TYPE ST_St020_HMI_IN_OUT : // EXTENDS ST_HMI_TR_CMD :
STRUCT
END_STRUCT
END_TYPE

(* stored: Version 1.1.0.1
   DUT ST_St020_HMI_IN_OUT: Id {35e7b9fa-7b10-4638-aa48-d58869c2fd85} *)
